(* IEC 61131-3 sources: AX-Repository/src, 2 files *)

(* ---- library.st ---- *)
//USING AxUnit;
NAMESPACE MotorClass

    CLASS PUBLIC Motor
        VAR PRIVATE
            _started : BOOL;
            _ended : BOOL;
        END_VAR

        VAR PUBLIC
            isRunning : BOOL;
        END_VAR

        METHOD PUBLIC Start : BOOL
            VAR_INPUT
                _proceed: BOOL;
            END_VAR
            IF _proceed AND NOT isRunning THEN
                _started:= TRUE;
                _ended := NOT _started;
                isRunning := _started;
                Start := _started;
            END_IF;
        END_METHOD

        METHOD PUBLIC Stop : BOOL
            VAR_INPUT
            _proceed: BOOL;
            END_VAR
            IF _proceed AND isRunning THEN
                _started:= FALSE;
                _ended := NOT _started;
                isRunning:=_started;
                Stop := _ended;
            END_IF;
        END_METHOD

        METHOD PUBLIC Invert : BOOL
            VAR_INPUT
                _proceed: BOOL;
            END_VAR
            IF _proceed THEN
             isRunning := NOT isRunning;
            END_IF;
            Invert := isRunning; //Invert vale come ouptup bool, devo togliere :BOOL per ottenere una void
        END_METHOD
    END_CLASS
/*
    {TestFixture}
    CLASS MotorBehaviorTests

        VAR PROTECTED
            testInstance : Motor;
        END_VAR

        {Test} //PRAGMAS - etichette nel codice
        METHOD PUBLIC StartBehaviorTest
            VAR_TEMP
                result : BOOL;
            END_VAR

            result := testInstance.Start();

            Assert.Equal(actual := result, expected := FALSE);

        END_METHOD
    END_CLASS
    */
END_NAMESPACE

(* ---- wrapper.st ---- *)
//USING MotorClass;
USING Siemens.Simatic.S71500.Clocks;

NAMESPACE MotorLibrary

    FUNCTION_BLOCK MotorWrapper
        VAR_INPUT
            abilita : BOOL;
        END_VAR
        VAR_OUTPUT
            risultato : BOOL;
        END_VAR
        VAR
            m : MotorClass.Motor;
        END_VAR

            risultato := m.Invert(_proceed:=abilita);

    END_FUNCTION_BLOCK

   /* FUNCTION_BLOCK FunzioneCounter
        VAR_INPUT
            a : INT;
            b : INT;
            aumenta : BOOL;
            diminuisci : BOOL;
            resetta : BOOL;
        END_VAR
        VAR
            s : INT;
            myCounter : Counter;
        END_VAR
        VAR_OUTPUT
            outadd : INT;
            outcount : LINT;
            resCount : LINT;
        END_VAR
        myCounter(up := aumenta, down := diminuisci, reset:= resetta, value => outcount);
        outadd := a + b;
    END_FUNCTION_BLOCK
    */

    FUNCTION_BLOCK FunzioneClock
        VAR
            measurement : RuntimeMeasurement;
            inSeconds : LREAL;
            started : BOOL;
        END_VAR
        VAR_INPUT
            a : INT;
            b : INT;
            aumenta : BOOL;
            diminuisci : BOOL;
        END_VAR
        VAR_OUTPUT
            outadd : INT;
        END_VAR
        IF aumenta AND NOT started THEN
            measurement.Start();
            started:= TRUE;
        ELSIF aumenta THEN
            inSeconds:=measurement.GetElapsedSeconds();
        ELSE
            measurement.Stop();
            started:=FALSE;
        END_IF;
        IF inSeconds>5 AND inSeconds<30 THEN
            outadd := a + outadd;
        ELSIF inSeconds>30 THEN
            measurement.Stop();
            started:=FALSE;
        END_IF;
    END_FUNCTION_BLOCK

END_NAMESPACE
